(* Logix 5000 project; controller Todd_Test vendor 1 type 14 code 87 rev 20.19; software revision 20.04 *)

TASK MainTask (continuous, watchdog 500 ms) : MainProgram

MODULES
   Controller : vendor 1 type 14 code 87 (CompactLogixL23E_QB1_Controller 0, rev 20.19)
      LocalENB : vendor 1 type 12 code 190 (CompactLogixL23E_QB1_Ethernet 1, rev 20.11)
      Local : CompactBus (CompactVirtualAdapter 3, rev 20.11)
         Discrete_Inputs : vendor 1 type 7 code 320 (Compact 1, rev 3.1, Input RPI 20 ms)
         Discrete_Outputs : vendor 1 type 7 code 322 (Compact 2, rev 3.1, Output RPI 20 ms)
END_MODULES

TYPE ac_JobData :
STRUCT
   NoOperation : BOOL;
   Valid : BOOL;
   Invalid : BOOL;
   MisMatch : BOOL;
   Prompt : BOOL;
   OneShot : INT;
   Offset : DINT;
   HMIOffsetSelect : DINT;
   PartCode : DINT;
   License_Batch : STRING;
   Enable : z_HMIStylePBs;
   Data : z_Data;
END_STRUCT
END_TYPE

TYPE BEP_BS1 :
STRUCT
   License_Batch : STRING;
   PartCode : DINT;
   Handshake : DINT;
   FaultStatus : DINT;
END_STRUCT
END_TYPE

TYPE BS1_BEP :
STRUCT
   License_Batch : STRING;
   Type_ID : DINT;
   Handshake : DINT;
   FaultStatus : DINT;
END_STRUCT
END_TYPE

TYPE dt_Data_Track :
STRUCT
   DataGT0 : BOOL;
   PPCurrent : BOOL;
   NPPCurrent : BOOL;
   PEN : BOOL;
   NEQPrev : BOOL;
   MDTBuffer : BOOL;
   MDTNext : BOOL;
   Move : BOOL;
   MoveDat2PRev : BOOL;
   Move0toNext : BOOL;
   InputWord : DINT;
   OutputWord : DINT;
END_STRUCT
END_TYPE

TYPE dt_DataTrack :
STRUCT
   NoProc : BOOL;
   NoParts : BOOL;
   NoData : BOOL;
END_STRUCT
END_TYPE

TYPE dt_Prelims :
STRUCT
   BuffDat : BOOL;
   InitDat : BOOL;
   StaDat : BOOL;
   PrevDat : BOOL;
   NextDat : BOOL;
   MTBuff : BOOL;
END_STRUCT
END_TYPE

TYPE int_FromConveyor :
STRUCT
   Hearbeat : BOOL;
   PartPresent : BOOL;
   DataPresent : BOOL;
   CleartoExit : BOOL;
   BypassPart : BOOL;
   ComsGood : BOOL;
   SpareBool_2 : BOOL;
   SpareBool_3 : BOOL;
   SpareBool_4 : BOOL;
   PartCode : DINT;
   SpareDINT : DINT;
END_STRUCT
END_TYPE

TYPE int_ToConveyor :
STRUCT
   Heartbeat : BOOL;
   ReadytoReceiveAssembly : BOOL;
   ReadytoReceivePartCode : BOOL;
   PartCodeReceived : BOOL;
   PartReceivedACK : BOOL;
   ReadytoExit : BOOL;
   GoodPart : BOOL;
   RejectPart : BOOL;
   Partpresent_1 : BOOL;
   Partpresent_2 : BOOL;
   Partpresent_3 : BOOL;
   comsgood : BOOL;
   AutoMode : BOOL;
   ManualMode : BOOL;
   SpareBool_4 : BOOL;
   LastPart : DINT;
   CurrentPart : DINT;
END_STRUCT
END_TYPE

TYPE PF52x_I :
STRUCT
   DriveStatus : INT;
   Ready : BOOL;
   Active : BOOL;
   CommandDir : BOOL;
   ActualDir : BOOL;
   Accelerating : BOOL;
   Decelerating : BOOL;
   Faulted : BOOL;
   AtReference : BOOL;
   CommFreqCnt : BOOL;
   CommLogicCnt : BOOL;
   ParmsLocked : BOOL;
   DigIn1Active : BOOL;
   DigIn2Active : BOOL;
   DigIn3Active : BOOL;
   DigIn4Active : BOOL;
   OutputFreq : INT;
END_STRUCT
END_TYPE

TYPE PF52x_O :
STRUCT
   LogicCommand : INT;
   Stop : BOOL;
   Start : BOOL;
   Jog : BOOL;
   ClearFaults : BOOL;
   Forward : BOOL;
   Reverse : BOOL;
   ForceKeypadCtrl : BOOL;
   MOPIncrement : BOOL;
   AccelRate1 : BOOL;
   AccelRate2 : BOOL;
   DecelRate1 : BOOL;
   DecelRate2 : BOOL;
   FreqSel01 : BOOL;
   FreqSel02 : BOOL;
   FreqSel03 : BOOL;
   MOPDecrement : BOOL;
   FreqCommand : INT;
END_STRUCT
END_TYPE

TYPE u_AccuracyBalanceSequence :
STRUCT
   SpinCount : COUNTER;
   ReSpinDwell : TIMER;
   SequenceStep : u_TireBalanceAccuracySteps;
   OneShot : BOOL[32];
END_STRUCT
END_TYPE

TYPE u_ActionAdvanceReturn :
STRUCT
   Advance : up_ActionNew;
   Return : up_ActionNew;
END_STRUCT
END_TYPE

TYPE u_ActionCloseOpen :
STRUCT
   Close : up_ActionNew;
   Open : up_ActionNew;
END_STRUCT
END_TYPE

TYPE u_ActionEngDiseng :
STRUCT
   Engage : up_ActionNew;
   Disengage : up_ActionNew;
END_STRUCT
END_TYPE

TYPE u_ActionInflate :
STRUCT
   Comp : BOOL;
   ProcComp : BOOL;
   Auto : BOOL;
   AutoSetup : BOOL;
   Clear : BOOL;
   ClrSetup : BOOL;
   OutPwr : BOOL;
   Cmd : BOOL;
   Out : BOOL;
   Mem : BOOL;
   PB : BOOL;
   FLT : BOOL;
   Active : BOOL;
   EnableSkip : BOOL;
   EnableBypass : BOOL;
   Bypassed : BOOL;
   Prompt : BOOL;
   OutPwrPrompt : BOOL;
   AtBeadSeat : BOOL;
   BeadSeatProcessComp : BOOL;
   Setup3 : BOOL;
   Setup4 : BOOL;
   AntiRept : BOOL;
   OneShot : BOOL;
   Text : DINT;
   StatusType : DINT;
   SeatTMR : TIMER;
   FaultTMR : TIMER;
   TestTMR : TIMER;
END_STRUCT
END_TYPE

TYPE u_ActionInflateDeflate :
STRUCT
   Inflate : u_ActionInflate;
   Deflate : up_ActionNew;
END_STRUCT
END_TYPE

TYPE u_ActionInOut :
STRUCT
   In : up_ActionNew;
   Out : up_ActionNew;
END_STRUCT
END_TYPE

TYPE u_ActionLower4Raise :
STRUCT
   LowerToLock : up_ActionNew;
   LowerToChanger : up_ActionNew;
   LowerToJoin_1 : up_ActionNew;
   LowerToJoin_2 : up_ActionNew;
   Raise : up_ActionNew;
END_STRUCT
END_TYPE

TYPE u_ActionRaiseLower :
STRUCT
   Raise : up_ActionNew;
   Lower : up_ActionNew;
END_STRUCT
END_TYPE

TYPE u_ActionRetractExtend :
STRUCT
   Retract : up_ActionNew;
   Extend : up_ActionNew;
END_STRUCT
END_TYPE

TYPE u_BalanceGainCalSeq :
STRUCT
   SequenceStep : u_TireBalanceGainSteps;
   OneShot : BOOL[32];
END_STRUCT
END_TYPE

TYPE u_BalanceToolingCalibrationSequence :
STRUCT
   SequenceStep : u_TireBalanceToolCalSteps;
   OneShot : BOOL[32];
   CycleCounter : COUNTER;
   IndexAngle : REAL;
END_STRUCT
END_TYPE

TYPE u_StaMode :
STRUCT
   AutoReqAntiRpt : BOOL;
   AutoRdy : BOOL;
   Auto : BOOL;
   ExtrnAutoRdy : BOOL;
   Man : BOOL;
   Calibration : BOOL;
   ByPass : BOOL;
   BatchMode : BOOL;
   Tryout : BOOL;
END_STRUCT
END_TYPE

TYPE u_StaMode_BeadSeat :
STRUCT
   AutoReqAntiRpt : BOOL;
   AutoRdy : BOOL;
   Auto : BOOL;
   ExtrnAutoRdy : BOOL;
   Man : BOOL;
   TryOut : BOOL;
   ByPass : BOOL;
END_STRUCT
END_TYPE

TYPE u_TBAL_BALCycle :
STRUCT
   Action : up_ActionNew;
   Seq : u_TBAL_BALSteps;
   ChargeAmpDwell : TIMER;
   SampleDelay : TIMER;
   SpinDwell : TIMER;
   ChargeAmp : up_Relay;
   OneShot : BOOL[32];
END_STRUCT
END_TYPE

TYPE u_TBAL_BALSteps :
STRUCT
   EnableChargeAmplifier : BOOL;
   StartRotation : BOOL;
   SpindleAtSpeed : BOOL;
   StartSample : BOOL;
   SampleComplete : BOOL;
   StopAtAngle : BOOL;
   CorrectStopPosition : BOOL;
   CycleComplete : BOOL;
END_STRUCT
END_TYPE

TYPE u_TireBalanceAccuracySteps :
STRUCT
   CloseCentering : BOOL;
   LowerLifter : BOOL;
   OpenCentering : BOOL;
   LowerUpperTooling : BOOL;
   LockLowerTooling : BOOL;
   UnlockUpperTooling : BOOL;
   InflateTire : BOOL;
   PromptForEmptySpin : BOOL;
   StartBalanceEmpty : BOOL;
   PromptOpenDoorCouple : BOOL;
   PromptCoupleWeights : BOOL;
   PromptCoupleSpin : BOOL;
   StartCoupleSpin : BOOL;
   PromptOpenDoorStatic : BOOL;
   PrmptStaticWeights : BOOL;
   PromptForStaticSpin : BOOL;
   StartStaticSpin : BOOL;
   PromptOpenDoorLower : BOOL;
   PromptLowerWeight : BOOL;
   PromptForLowerSpin : BOOL;
   StartLowerSpin : BOOL;
   PromptOpenDoorUpper : BOOL;
   PromptUpperWeight : BOOL;
   PromptForUpperSpin : BOOL;
   StartUpperSpin : BOOL;
   PromptRemoveWeights : BOOL;
   PromptTestComplete : BOOL;
   DeflateTire : BOOL;
   LockUpperTooling : BOOL;
   ExtendBeadBreaker : BOOL;
   UnlockLowerTooling : BOOL;
   RaiseUpperTooling : BOOL;
   RaiseLifter : BOOL;
   RaiseBeadBreaker : BOOL;
   AccuracyTestComplete : BOOL;
END_STRUCT
END_TYPE

TYPE u_TireBalanceGainSteps :
STRUCT
   CloseCentering : BOOL;
   LowerLifter : BOOL;
   OpenCentering : BOOL;
   LowerUpperTooling : BOOL;
   LockLowerTooling : BOOL;
   UnlockUpperTooling : BOOL;
   InflateTire : BOOL;
   PromptForEmptySpin : BOOL;
   StartBalanceEmpty : BOOL;
   PromptOpenDoorUpper : BOOL;
   PromptUpperWeight : BOOL;
   PromptForUpperSpin : BOOL;
   StartBalanceUpper : BOOL;
   PromptOpenDoorLower : BOOL;
   PromptLowerWeight : BOOL;
   PromptForLowerSpin : BOOL;
   StartBalanceLower : BOOL;
   PromptOpenDoorEmpty : BOOL;
   PromptRemoveWeights : BOOL;
   DeflateTire : BOOL;
   LockUpperTooling : BOOL;
   ExtendBeadBreakers : BOOL;
   UnlockLowerTooling : BOOL;
   RaiseUpperTooling : BOOL;
   RaiseLifter : BOOL;
   RaiseBeadBreakers : BOOL;
   GainCalibrationComplete : BOOL;
END_STRUCT
END_TYPE

TYPE u_TireBalanceToolCalSteps :
STRUCT
   CloseCentering : BOOL;
   LowerLifter : BOOL;
   OpenCentering : BOOL;
   LowerUpperTooling : BOOL;
   LockLowerTooling : BOOL;
   UnlockUpperTooling : BOOL;
   InflateTire : BOOL;
   StartBalance : BOOL;
   DeflateTire : BOOL;
   LockUpperTooling : BOOL;
   AdvanceBeadBreakers : BOOL;
   UnlockLowerTooling : BOOL;
   RaiseUpperTooling : BOOL;
   IndexTireToNextAngle : BOOL;
   RaiseLifter : BOOL;
   RaiseBeadBreaker : BOOL;
   AlignTooling : BOOL;
END_STRUCT
END_TYPE

TYPE uc_BDS_XFRIntlk :
STRUCT
   Auto : BOOL;
   Man : BOOL;
   AtLoad : BOOL;
   AtUnload : BOOL;
   Bypass : BOOL;
   ByPassAllowed : BOOL;
   InPosition : BOOL;
   NextConvFull : BOOL;
   LeavingPX : BOOL;
   Load_Unload : BOOL;
   DriveOK : BOOL;
   HiSpdEn : BOOL;
   DrvRunningFwd : BOOL;
   DrvRunningRev : BOOL;
   TWRunAudit : BOOL;
   PrimaryBalanceMode : BOOL;
   RdytoExitFwd : BOOL;
   RdytoExitRev : BOOL;
   RdytoExitSide : BOOL;
   RequestNextPart : BOOL;
   ClrtoEnterFwd : BOOL;
   ClrtoEnterRev : BOOL;
   ClrtoEnterSide : BOOL;
   JobinTransitFwd : BOOL;
   JobinTransitRev : BOOL;
   JobinTransitSide : BOOL;
   IndexInPB : BOOL;
   IndexOutPB : BOOL;
   RevInPB : BOOL;
   RevOutPB : BOOL;
   BalanceSampleComplete : BOOL;
   ValidModel : BOOL;
   MachineEmpty : BOOL;
   NoSkidPres : BOOL;
   Heartbeat : BOOL;
END_STRUCT
END_TYPE

TYPE uc_BeadSeaterServoTargets :
STRUCT
   PressUnitAdvanced : REAL;
   PressUnitReturned : REAL;
   UpperUnitAdvanced : REAL;
   LowerUnitAdvanced : REAL;
   UpperRollerAdvanced : REAL;
   LowerRollerAdvanced : REAL;
   LifterMidPosition : REAL;
   LifterLowerPosition : REAL;
END_STRUCT
END_TYPE

TYPE uc_BeadSeaterServoTargetsWithTorque :
STRUCT
   PressUnitAdvanced : REAL;
   PressUnitReturned : REAL;
   UpperUnitAdvanced : REAL;
   LowerUnitAdvanced : REAL;
   UpperRollerAdvanced : REAL;
   UpperRollerAdvanceLowTorqueLimit : REAL;
   UpperRollerAdvanceHighTorqueLimit : REAL;
   UpperRollerAdvanceMinTorqueApplied : REAL;
   UpperRollerAdvanceMaxTorqueApplied : REAL;
   LowerRollerAdvanced : REAL;
   LowerRollerAdvanceLowTorqueLimit : REAL;
   LowerRollerAdvanceHighTorqueLimit : REAL;
   LowerRollerAdvanceMinTorqueApplied : REAL;
   LowerRollerAdvanceMaxTorqueApplied : REAL;
   LifterMidPosition : REAL;
   LifterLowerPosition : REAL;
END_STRUCT
END_TYPE

TYPE uc_Gripper :
STRUCT
   GripTorque : REAL;
   GripSpeed : REAL;
   RelaxSpeed : REAL;
   RelaxOffset : REAL;
END_STRUCT
END_TYPE

TYPE uc_Home :
STRUCT
   HomingTorque : REAL;
   Offset : REAL;
   Velocity : REAL;
END_STRUCT
END_TYPE

TYPE uc_Job :
STRUCT
   TWStatus : uc_TWStatus;
   TWModel : uc_TWModel;
   TWCorrection : uc_TWCorrection;
   Xfer : uc_BDS_XFRIntlk;
END_STRUCT
END_TYPE

TYPE uc_Job_BC :
STRUCT
   TWStatus : uc_TWStatus;
   TWModel : uc_TWModel;
   TWCorrection : uc_TWCorrection;
   Xfer : uc_BDS_XFRIntlk;
   BarCode : SINT[80];
END_STRUCT
END_TYPE

TYPE uc_KokusaiModelData :
STRUCT
   Name : STRING;
   WheelDiam : DINT;
   WheelWidth : DINT;
   WheelOffset : DINT;
   OutsideDiameter : DINT;
   PressStroke : DINT;
   Bypass : BOOL;
   Servo : uc_BeadSeaterServoTargets;
   RotateTime : DINT;
END_STRUCT
END_TYPE

TYPE uc_KokusaiModelDataWithTorque :
STRUCT
   Type_ID : DINT;
   WheelDiam : DINT;
   WheelWidth : DINT;
   WheelOffset : DINT;
   OutsideDiameter : REAL;
   PressStroke : DINT;
   Bypass : BOOL;
   Servo : uc_BeadSeaterServoTargetsWithTorque;
   RotateTime : DINT;
END_STRUCT
END_TYPE

TYPE uc_KokusaiModelTorqueData :
STRUCT
   LowerRollerAdvanceTorqueApplied : REAL[101];
   LowerRollerRotatingMinTorqueApplied : REAL[101];
   LowerRollerRotatingMaxTorqueApplied : REAL[101];
   LowerRollerRotatingAveTorqueApplied : REAL[101];
   UpperRollerAdvanceTorqueApplied : REAL[101];
   UpperRollerRotatingMinTorqueApplied : REAL[101];
   UpperRollerRotatingMaxTorqueApplied : REAL[101];
   UpperRollerRotatingAveTorqueApplied : REAL[101];
END_STRUCT
END_TYPE

TYPE uc_TransferInterlock :
STRUCT
   Auto : BOOL;
   Man : BOOL;
   AtLoad : BOOL;
   AtUnload : BOOL;
   Bypass : BOOL;
   InPosition : BOOL;
   NextConvFull : BOOL;
   LeavingPX : BOOL;
   Spare8 : BOOL;
   DriveOK : BOOL;
   HiSpdEn : BOOL;
   DrvRunningFwd : BOOL;
   DrvRunningRev : BOOL;
   Spare13 : BOOL;
   Spare14 : BOOL;
   RdytoExitFwd : BOOL;
   RdytoExitRev : BOOL;
   RdytoExitSide : BOOL;
   ClrtoEnterFwd : BOOL;
   ClrtoEnterRev : BOOL;
   ClrtoEnterSide : BOOL;
   JobinTransitFwd : BOOL;
   JobinTransitRev : BOOL;
   JobinTransitSide : BOOL;
   IndexInPB : BOOL;
   IndexOutPB : BOOL;
   RevInPB : BOOL;
   RevOutPB : BOOL;
   Spare28 : BOOL;
   Spare29 : BOOL;
   MachineEmpty : BOOL;
   NoSkidPres : BOOL;
   Heartbeat : DINT;
   BEP_BS1_ComboRdyToReceive : BOOL;
   BEP_BS1_ComboReceived : BOOL;
   BEP_BS1_ComboDataMismatch : BOOL;
   BEP_BS1_BypassStation : BOOL;
   BEP_BS1_RejectAssy : BOOL;
   BS1_BEP_ComboSent : BOOL;
   BS1_BEP_ComboReceived : BOOL;
   BS1_BEP_NotTested : BOOL;
   BS1_BEP_PartPresent : BOOL;
   BS1_BEP_ComboDataMismatch : BOOL;
   BS1_BEP_CheckTireMode : BOOL;
   ComboRdyToReceive : BOOL;
END_STRUCT
END_TYPE

TYPE uc_TransferInterlock_New :
STRUCT
   Auto : BOOL;
   Man : BOOL;
   AtLoad : BOOL;
   AtUnload : BOOL;
   Bypass : BOOL;
   InPosition : BOOL;
   NextConvFull : BOOL;
   LeavingPX : BOOL;
   AdapterOKForNext : BOOL;
   DriveOK : BOOL;
   HiSpdEn : BOOL;
   DrvRunningFwd : BOOL;
   DrvRunningRev : BOOL;
   AdapterOKForCurrent : BOOL;
   RequestNextPart : BOOL;
   RdytoExitFwd : BOOL;
   RdytoExitRev : BOOL;
   RdytoExitSide : BOOL;
   TransferedDataFwd : BOOL;
   TransferedDataRev : BOOL;
   TransferedDataSide : BOOL;
   ClrToEnterFwd : BOOL;
   ClrToEnterRev : BOOL;
   ClrToEnterSide : BOOL;
   JobinTransitFwd : BOOL;
   JobinTransitRev : BOOL;
   JobinTransitSide : BOOL;
   IndexInPB : BOOL;
   IndexOutPB : BOOL;
   RevInPB : BOOL;
   RevOutPB : BOOL;
   Spare28 : BOOL;
   Spare29 : BOOL;
   Spare30 : BOOL;
   NoSkidPres : BOOL;
   Heartbeat : DINT;
END_STRUCT
END_TYPE

TYPE uc_TWCorrection :
STRUCT
   BalanceStaticAmount : REAL;
   BalanceStaticAngle : DINT;
   BalanceCoupleAmount : REAL;
   BalanceCoupleAngle : DINT;
   PlaneUpperAmount : REAL;
   PlaneUpperAngle : DINT;
   PlaneLowerAmount : REAL;
   PlaneLowerAngle : DINT;
   UpperWeightAmount : REAL;
   UpperWeightAngle : DINT;
   UpperWeightStyle : DINT;
   LowerWeightAmount : REAL;
   LowerWeightAngle : DINT;
   LowerWeightStyle : DINT;
   ShortReachCorrection : DINT;
   SecondCorrection : DINT;
   FirstCorrection : DINT;
   UpperWeightRadius : DINT;
   LowerWeightRadius : DINT;
   UpperWeightHeight : DINT;
   LowerWeightHeight : DINT;
END_STRUCT
END_TYPE

TYPE uc_TWModel :
STRUCT
   PartCode : DINT;
   WheelDiameter : DINT;
   Desc0_1 : DINT;
   Desc2_3 : DINT;
   Desc4_5 : DINT;
   Desc6_7 : DINT;
   Desc8_9 : DINT;
   Desc10_11 : DINT;
   Desc12_13 : DINT;
   Desc14_15 : DINT;
   Desc16_17 : DINT;
   Desc18_19 : DINT;
   Key : DINT;
   TID : DINT;
END_STRUCT
END_TYPE

TYPE uc_TWStatus :
STRUCT
   GoodAssembly : BOOL;
   CorrectableAssembly : BOOL;
   UncorrectableAssembly : BOOL;
   ByPassAssembly : BOOL;
   MiniSpare : BOOL;
   Material : BOOL;
   MidPlaneApply : BOOL;
   UpSideDown : BOOL;
END_STRUCT
END_TYPE

TYPE uc_UFB_BALData :
STRUCT
   Rank : INT;
   MarkPattern : INT;
   SortPosition : INT;
   MarkAngle : INT;
   StaticAmount : REAL;
   StaticAmountUnits : INT;
   StaticAngle : INT;
   CoupleAmount : REAL;
   CoupleAmountUnits : INT;
   CoupleAngle : INT;
   UpperAmount : REAL;
   UpperAmountUnits : INT;
   UpperAngle : INT;
   LowerAmount : REAL;
   LowerAmountUnits : INT;
   LowerAngle : INT;
END_STRUCT
END_TYPE

TYPE uc_UFB_BALStatus :
STRUCT
   ByPass : BOOL;
   BALGainCalRequired : BOOL;
   BALToolCalRequired : BOOL;
   MeasureBAL : BOOL;
END_STRUCT
END_TYPE

TYPE uc_UFB_Data :
STRUCT
   Model : INT;
   RimStep : INT;
   Adapter : INT;
   BeadDiameter : INT;
   BeadWidth : INT;
   OutsideDiameter : INT;
   Weight : INT;
   RankFinal : INT;
   MarkPatternFinal : INT;
   SortPositionFinal : INT;
   SerialNumber : SINT[20];
   BAL : uc_UFB_BALData;
   RO : uc_UFB_ROData;
   LSU : uc_UFB_LSUData;
   HSU : uc_UFB_HSUData;
END_STRUCT
END_TYPE

TYPE uc_UFB_HSUData :
STRUCT
   Rank : INT;
   MarkPattern : INT;
   SortPosition : INT;
   MarkAngle : INT;
   LoadForce : INT;
   ConicityForce : INT;
   PlySteerForce : INT;
   SpeedRPM : INT;
   SurfaceVelocity : INT;
   RadialOverallAmountCW : INT;
   RadialOverallAngleCW : INT;
   Radial1stHarmonicAmountCW : INT;
   Radial1stHarmonicAngleCW : INT;
   Radial2ndHarmonicAmountCW : INT;
   Radial2ndHarmonicAngleCW : INT;
   Radial3rdHarmonicAmountCW : INT;
   Radial3rdHarmonicAngleCW : INT;
   Radial4thHarmonicAmountCW : INT;
   Radial4thHarmonicAngleCW : INT;
   Radial5thHarmonicAmountCW : INT;
   Radial5thHarmonicAngleCW : INT;
   RadialOverallAmountCCW : INT;
   RadialOverallAngleCCW : INT;
   Radial1stHarmonicAmountCCW : INT;
   Radial1stHarmonicAngleCCW : INT;
   Radial2ndHarmonicAmountCCW : INT;
   Radial2ndHarmonicAngleCCW : INT;
   Radial3rdHarmonicAmountCCW : INT;
   Radial3rdHarmonicAngleCCW : INT;
   Radial4thHarmonicAmountCCW : INT;
   Radial4thHarmonicAngleCCW : INT;
   Radial5thHarmonicAmountCCW : INT;
   Radial5thHarmonicAngleCCW : INT;
   LateralOverallAmountCW : INT;
   LateralOverallAngleCW : INT;
   Lateral1stHarmonicAmountCW : INT;
   Lateral1stHarmonicAngleCW : INT;
   Lateral2ndHarmonicAmountCW : INT;
   Lateral2ndHarmonicAngleCW : INT;
   Lateral3rdHarmonicAmountCW : INT;
   Lateral3rdHarmonicAngleCW : INT;
   Lateral4thHarmonicAmountCW : INT;
   Lateral4thHarmonicAngleCW : INT;
   Lateral5thHarmonicAmountCW : INT;
   Lateral5thHarmonicAngleCW : INT;
   LateralForceDeviationAmountCW : INT;
   LateralOverallAmountCCW : INT;
   LateralOverallAngleCCW : INT;
   Lateral1stHarmonicAmountCCW : INT;
   Lateral1stHarmonicAngleCCW : INT;
   Lateral2ndHarmonicAmountCCW : INT;
   Lateral2ndHarmonicAngleCCW : INT;
   Lateral3rdHarmonicAmountCCW : INT;
   Lateral3rdHarmonicAngleCCW : INT;
   Lateral4thHarmonicAmountCCW : INT;
   Lateral4thHarmonicAngleCCW : INT;
   Lateral5thHarmonicAmountCCW : INT;
   Lateral5thHarmonicAngleCCW : INT;
   LateralForceDeviationAmountCCW : INT;
   TangentialOverallAmountCW : INT;
   TangentialOverallAngleCW : INT;
   Tangential1stHarmonicAmountCW : INT;
   Tangential1stHarmonicAngleCW : INT;
   Tangential2ndHarmonicAmountCW : INT;
   Tangential2ndHarmonicAngleCW : INT;
   Tangential3rdHarmonicAmountCW : INT;
   Tangential3rdHarmonicAngleCW : INT;
   Tangential4thHarmonicAmountCW : INT;
   Tangential4thHarmonicAngleCW : INT;
   Tangential5thHarmonicAmountCW : INT;
   Tangential5thHarmonicAngleCW : INT;
   TangentialOverallAmountCCW : INT;
   TangentialOverallAngleCCW : INT;
   Tangential1stHarmonicAmountCCW : INT;
   Tangential1stHarmonicAngleCCW : INT;
   Tangential2ndHarmonicAmountCCW : INT;
   Tangential2ndHarmonicAngleCCW : INT;
   Tangential3rdHarmonicAmountCCW : INT;
   Tangential3rdHarmonicAngleCCW : INT;
   Tangential4thHarmonicAmountCCW : INT;
   Tangential4thHarmonicAngleCCW : INT;
   Tangential5thHarmonicAmountCCW : INT;
   Tangential5thHarmonicAngleCCW : INT;
END_STRUCT
END_TYPE

TYPE uc_UFB_Job :
STRUCT
   Data : uc_UFB_Data;
   Status : uc_UFB_Status;
END_STRUCT
END_TYPE

TYPE uc_UFB_LSUData :
STRUCT
   Rank : INT;
   MarkPattern : INT;
   SortPosition : INT;
   MarkAngle : INT;
   LoadForce : INT;
   ConicityForce : INT;
   PlySteerForce : INT;
   SpeedRPM : INT;
   SurfaceVelocity : INT;
   RadialOverallAmountCW : INT;
   RadialOverallAngleCW : INT;
   Radial1stHarmonicAmountCW : INT;
   Radial1stHarmonicAngleCW : INT;
   Radial2ndHarmonicAmountCW : INT;
   Radial2ndHarmonicAngleCW : INT;
   Radial3rdHarmonicAmountCW : INT;
   Radial3rdHarmonicAngleCW : INT;
   Radial4thHarmonicAmountCW : INT;
   Radial4thHarmonicAngleCW : INT;
   Radial5thHarmonicAmountCW : INT;
   Radial5thHarmonicAngleCW : INT;
   RadialOverallAmountCCW : INT;
   RadialOverallAngleCCW : INT;
   Radial1stHarmonicAmountCCW : INT;
   Radial1stHarmonicAngleCCW : INT;
   Radial2ndHarmonicAmountCCW : INT;
   Radial2ndHarmonicAngleCCW : INT;
   Radial3rdHarmonicAmountCCW : INT;
   Radial3rdHarmonicAngleCCW : INT;
   Radial4thHarmonicAmountCCW : INT;
   Radial4thHarmonicAngleCCW : INT;
   Radial5thHarmonicAmountCCW : INT;
   Radial5thHarmonicAngleCCW : INT;
   LateralOverallAmountCW : INT;
   LateralOverallAngleCW : INT;
   Lateral1stHarmonicAmountCW : INT;
   Lateral1stHarmonicAngleCW : INT;
   Lateral2ndHarmonicAmountCW : INT;
   Lateral2ndHarmonicAngleCW : INT;
   Lateral3rdHarmonicAmountCW : INT;
   Lateral3rdHarmonicAngleCW : INT;
   Lateral4thHarmonicAmountCW : INT;
   Lateral4thHarmonicAngleCW : INT;
   Lateral5thHarmonicAmountCW : INT;
   Lateral5thHarmonicAngleCW : INT;
   LateralForceDeviationAmountCW : INT;
   LateralOverallAmountCCW : INT;
   LateralOverallAngleCCW : INT;
   Lateral1stHarmonicAmountCCW : INT;
   Lateral1stHarmonicAngleCCW : INT;
   Lateral2ndHarmonicAmountCCW : INT;
   Lateral2ndHarmonicAngleCCW : INT;
   Lateral3rdHarmonicAmountCCW : INT;
   Lateral3rdHarmonicAngleCCW : INT;
   Lateral4thHarmonicAmountCCW : INT;
   Lateral4thHarmonicAngleCCW : INT;
   Lateral5thHarmonicAmountCCW : INT;
   Lateral5thHarmonicAngleCCW : INT;
   LateralForceDeviationAmountCCW : INT;
END_STRUCT
END_TYPE

TYPE uc_UFB_MEAStatus :
STRUCT
   ByPass : BOOL;
   ROToolCalRequired : BOOL;
   LSUToolCalRequired : BOOL;
   MeasureRO : BOOL;
   ROMeasureType : INT;
   MeasureLSU : BOOL;
   LSU_SingleDirection : BOOL;
   LSU_CWDirection : BOOL;
   EnglishUnits : BOOL;
END_STRUCT
END_TYPE

TYPE uc_UFB_ROData :
STRUCT
   Rank : INT;
   MarkPattern : INT;
   SortPosition : INT;
   MarkAngle : INT;
   RadialTopPeakAmount : INT;
   RadialTopPeakAngle : INT;
   RadialTop1stAmount : INT;
   RadialTop1stAngle : INT;
   RadialTop2ndAmount : INT;
   RadialTop2ndAngle : INT;
   RadialCenterPeakAmount : INT;
   RadialCenterPeakAngle : INT;
   RadialCenter1stAmount : INT;
   RadialCenter1stAngle : INT;
   RadialCenter2ndAmount : INT;
   RadialCenter2ndAngle : INT;
   RadialBottomPeakAmount : INT;
   RadialBottomPeakAngle : INT;
   RadialBottom1stAmount : INT;
   RadialBottom1stAngle : INT;
   RadialBottom2ndAmount : INT;
   RadialBottom2ndAngle : INT;
   LateralTopPeakAmount : INT;
   LateralTopPeakAngle : INT;
   LateralTop1stAmount : INT;
   LateralTop1stAngle : INT;
   LateralTop2ndAmount : INT;
   LateralTop2ndAngle : INT;
   LateralBottomPeakAmount : INT;
   LateralBottomPeakAngle : INT;
   LateralBottom1stAmount : INT;
   LateralBottom1stAngle : INT;
   LateralBottom2ndAmount : INT;
   LateralBottom2ndAngle : INT;
   TopBulgeAmount : INT;
   TopBulgeAngle : INT;
   TopDentAmount : INT;
   TopDentAngle : INT;
   BottomBulgeAmount : INT;
   BottomBulgeAngle : INT;
   BottomDentAmount : INT;
   BottomDentAngle : INT;
END_STRUCT
END_TYPE

TYPE uc_UFB_Status :
STRUCT
   ByPass : BOOL;
   CertificationMode : BOOL;
   UpSideDown : BOOL;
   MEA : uc_UFB_MEAStatus;
   BAL : uc_UFB_BALStatus;
END_STRUCT
END_TYPE

TYPE ud_KokusaiServoConstants :
STRUCT
   cForward : DINT;
   cReverse : DINT;
   cPercentMaxSpeed : DINT;
   cDisabled : DINT;
   cEnabled : DINT;
   cAbsolute : DINT;
   cIncremental : DINT;
   cRotaryShortestPath : DINT;
   cRotaryPositive : DINT;
   cRotaryNegative : DINT;
   cAbsoluteMasterOffset : DINT;
   cIncrementalMasterOffset : DINT;
   cTourqueLimit : ud_KokusaiServoTorqueContants;
END_STRUCT
END_TYPE

TYPE ud_KokusaiServoTorqueContants :
STRUCT
   Axis1 : REAL;
   Axis2 : REAL;
   Axis3 : REAL;
   Axis4 : REAL;
   Axis5 : REAL;
   Axis6 : REAL;
   Axis7 : REAL;
   Axis8 : REAL;
   Axis9 : REAL;
   Axis10 : REAL;
   Axis11 : REAL;
   Axis12 : REAL;
   Axis13 : REAL;
   Axis14 : REAL;
   Axis15 : REAL;
END_STRUCT
END_TYPE

TYPE ud_KokusaiTransferGripper :
STRUCT
   InPositionLowRangeLimit : DINT;
   InPositionHighRangeLimit : DINT;
   Model : ud_KokusaiTransferGripperModel[10000];
END_STRUCT
END_TYPE

TYPE ud_KokusaiTransferGripperModel :
STRUCT
   GripperClosedPositionHighSafety : DINT;
   GripperClosedPosition : REAL;
   GripperOpenedPositionHighSafety : DINT;
   GripperOpenedPosition : REAL;
END_STRUCT
END_TYPE

TYPE udt_AutomaticAutoStop :
STRUCT
   PP_CenteringConveyor : BOOL;
   PP_BeadSeaterStation : BOOL;
   Engaged : BOOL;
   Complete : BOOL;
   SpareBool_01 : BOOL;
   SpareBool_02 : BOOL;
   SpareBool_03 : BOOL;
   SpareBool_04 : BOOL;
   ONS : INT;
   SpareDint : DINT;
   EngageTimer : TIMER;
END_STRUCT
END_TYPE

TYPE udt_PanelViewButton :
STRUCT
   Enable_PVPB : BOOL;
   Enabled_PVLT : BOOL;
   EnabledInternal : BOOL;
   ONS : BOOL;
END_STRUCT
END_TYPE

TYPE up_ActionNew :
STRUCT
   Comp : BOOL;
   ProcComp : BOOL;
   Auto : BOOL;
   AutoSetup : BOOL;
   ClrSetup : BOOL;
   ClearStart : BOOL;
   ClearThru : BOOL;
   OutPwr : BOOL;
   Cmd : BOOL;
   Out : BOOL;
   Mem : BOOL;
   PB : BOOL;
   FLT : BOOL;
   Active : BOOL;
   EnableSkip : BOOL;
   EnableBypass : BOOL;
   Bypassed : BOOL;
   Prompt : BOOL;
   OutPwrPrompt : BOOL;
   Setup1 : BOOL;
   Setup2 : BOOL;
   Setup3 : BOOL;
   Setup4 : BOOL;
   AntiRept : BOOL;
   OneShot : BOOL[32];
   TMR : TIMER[5];
   FaultTMR : TIMER;
END_STRUCT
END_TYPE

TYPE up_BalanceLifter :
STRUCT
   Command : up_BalanceLifterCommands;
   Status : up_BalanceLifterStatus;
   MidPositionDwell : TIMER;
   EnableMotion : BOOL;
   RaiseTargetIsValid : BOOL;
   MiddleTargetIsValid : BOOL;
   LowerTargetIsValid : BOOL;
   RaisedPositionTarget : REAL;
   RaisedLowLimit : REAL;
   RaisedHighLimit : REAL;
   MiddlePositionTarget : REAL;
   MiddleLowLimit : REAL;
   MiddleHighLimit : REAL;
   MiddleLowSafety : REAL;
   MiddleHighSafety : REAL;
   LowerPositionTarget : REAL;
   LowerLowLimit : REAL;
   LowerHighLimit : REAL;
   LowerLowSafety : REAL;
   LowerHighSafety : REAL;
   JogSpeedPercent : DINT;
END_STRUCT
END_TYPE

TYPE up_BalanceLifterCommands :
STRUCT
   JogMode : BOOL;
   JogLifterDown : BOOL;
   JogLifterUp : BOOL;
   StartHomePulse : BOOL;
   HomeLifterServo : BOOL;
   SetLifterRaisedPosition : BOOL;
   SetLifterLoweredCalibration : BOOL;
   SetLifterMiddlePosition : BOOL;
   SetLifterLoweredPosition : BOOL;
END_STRUCT
END_TYPE

TYPE up_BalanceLifterStatus :
STRUCT
   AtHomePosition : BOOL;
   ValidRaisedPosition : BOOL;
   ValidMiddlePosition : BOOL;
   ValidLoweredPosition : BOOL;
END_STRUCT
END_TYPE

TYPE up_BalanceSpindleServo :
STRUCT
   Command : up_SpindleServoCommands;
   Status : up_SpindleServoStatus;
   EnableMotion : BOOL;
   StartHomeSearch : BOOL;
   SearchForSpindleHome : BOOL;
   RetrySetHome : BOOL;
   VelocityInRange : BOOL;
   AtBalanceSpeed : BOOL;
   AtRunoutSpeed : BOOL;
   RimChangeAngleValid : BOOL;
   RimUnlockAngleValid : BOOL;
   MarkerAngle : REAL;
   OrientTargetAngle : REAL;
   OrientTargetHighLimit : REAL;
   OrientTargetLowLimit : REAL;
   MaxVelocityError : REAL;
   UpperFaultSpeed : REAL;
   LowerFaultSpeed : REAL;
   UpperToolingAngle : REAL;
   UpperToolingHighLimit : REAL;
   UpperToolingLowLimit : REAL;
   UpperToolingAlignmentTarget : REAL;
   UpperToolingAlignmentError : REAL;
   JogSpeed : REAL;
   OrientSpeed : REAL;
   RunoutSpeed : REAL;
   RunoutSpeedHigh : REAL;
   RunoutSpeedLow : REAL;
   BalanceSpeed : REAL;
   BalanceSpeedHigh : REAL;
   BalanceSpeedLow : REAL;
   AccelRate : REAL;
   DecelRate : REAL;
   BalanceRevolutions : DINT;
   BalanceDistance : REAL;
   RunoutRevolutions : DINT;
   RunoutDistance : REAL;
   SpindleStartAngle : REAL;
   SpindleSlipAngle : REAL;
   FailsafeTimer : TIMER;
   RimChangerAngleTarget : REAL;
   RimChangerHighLimit : REAL;
   RimChangerLowLimit : REAL;
   RimChangeValidHighLimit : REAL;
   RimChangeValidLowLimit : REAL;
   RimUnlockAngleTarget : REAL;
   RimUnlockHighLimit : REAL;
   RimUnlockLowLimit : REAL;
   RimUnlockValidHighLimit : REAL;
   RimUnlockValidLowLimit : REAL;
END_STRUCT
END_TYPE

TYPE up_ConveyorServo :
STRUCT
   EnableMotion : BOOL;
   MoveInLength : REAL;
   MoveOutLength : REAL;
END_STRUCT
END_TYPE

TYPE up_ConveyorWidthServo :
STRUCT
   Command : up_ConveyorWidthServoCommands;
   Status : up_ConveyorWidthServoStatus;
   EnableMotion : BOOL;
   AdapterTargetValid : BOOL;
   TransferTargetValid : BOOL;
   AdapterPositionTarget : REAL;
   AdapterPositionHiLimit : REAL;
   AdapterPositionLoLimit : REAL;
   TransferPositionTarget : REAL;
   TransferPositionHiLimit : REAL;
   TransferPositionLoLimit : REAL;
   JogSpeedPercent : DINT;
END_STRUCT
END_TYPE

TYPE up_ConveyorWidthServoCommands :
STRUCT
   JogMode : BOOL;
   JogClose : BOOL;
   JogOpen : BOOL;
   StartHomePulse : BOOL;
   HomeServo : BOOL;
END_STRUCT
END_TYPE

TYPE up_ConveyorWidthServoStatus :
STRUCT
   HomePosition : BOOL;
   ValidAdapterPosition : BOOL;
   ValidTransferPosition : BOOL;
END_STRUCT
END_TYPE

TYPE up_Cycle :
STRUCT
   InCycle : BOOL;
   AllPartsLoaded : BOOL;
   Finished : BOOL;
   FirstAutoCycle : BOOL;
   LoadPosition : BOOL;
   NoPartsLoaded : BOOL;
   NoProcComp : BOOL;
   NoProcInit : BOOL;
   NoStepsComp : BOOL;
   ProcComp : BOOL;
   ResetProcComp : BOOL;
   Resume : BOOL;
   RetToLoad : BOOL;
   RetToUnload : BOOL;
   SetProcComp : BOOL;
   Start : BOOL;
   Started : BOOL;
   StepsComp : BOOL;
   UnLoadPosition : BOOL;
   WaitingForLoad : BOOL;
   Idle : TIMER;
END_STRUCT
END_TYPE

TYPE up_Cylinder :
STRUCT
   PX1 : BOOL;
   PX1NOnFlt : BOOL;
   PX1NOffFlt : BOOL;
   BypPX1NOn : BOOL;
   BypPX1NOff : BOOL;
   PX2 : BOOL;
   PX2NOnFlt : BOOL;
   PX2NOffFlt : BOOL;
   BypPX2NOn : BOOL;
   BypPX2NOff : BOOL;
END_STRUCT
END_TYPE

TYPE up_CylinderBackToBack :
STRUCT
   PX1 : BOOL;
   PX1NOnFlt : BOOL;
   PX1NOffFlt : BOOL;
   BypPX1NOn : BOOL;
   BypPX1NOff : BOOL;
   PX2 : BOOL;
   PX2NOnFlt : BOOL;
   PX2NOffFlt : BOOL;
   BypPX2NOn : BOOL;
   BypPX2NOff : BOOL;
   PX3 : BOOL;
   PX3NOnFlt : BOOL;
   PX3NOffFlt : BOOL;
   BypPX3NOn : BOOL;
   BypPX3NOff : BOOL;
   PX4 : BOOL;
   PX4NOnFlt : BOOL;
   PX4NOffFlt : BOOL;
   BypPX4NOn : BOOL;
   BypPX4NOff : BOOL;
END_STRUCT
END_TYPE

TYPE up_Motion5Position :
STRUCT
   PX1 : BOOL;
   PX2 : BOOL;
   PX3 : BOOL;
   PX4 : BOOL;
   PX5 : BOOL;
END_STRUCT
END_TYPE

TYPE up_Part :
STRUCT
   Pres : BOOL;
   NotPres : BOOL;
   PresSwitches : BOOL;
   NotPresSwitches : BOOL;
   PresMemory : BOOL;
   Sw1NotOff : BOOL;
   Sw2NotOff : BOOL;
   Sw3NotOff : BOOL;
   Sw4NotOff : BOOL;
   Sw5NotOff : BOOL;
   Sw6NotOff : BOOL;
   Sw1NotOn : BOOL;
   Sw2NotOn : BOOL;
   Sw3NotOn : BOOL;
   Sw4NotOn : BOOL;
   Sw5NotOn : BOOL;
   Sw6NotOn : BOOL;
   LoadedProp : BOOL;
   LoadPosn : BOOL;
   Load : up_ActionNew;
   TryoutPresent : TIMER;
   TryoutNotPresent : TIMER;
END_STRUCT
END_TYPE

TYPE up_Relay :
STRUCT
   DiagEnable : BOOL;
   FltedOnMem : BOOL;
   Input : BOOL;
   Mimic : BOOL;
   Output : BOOL;
   FltTim : TIMER;
   OnTim : TIMER;
END_STRUCT
END_TYPE

TYPE up_RunoutServo :
STRUCT
   Command : up_RunoutServoCommands;
   Status : up_RunoutServoStatus;
   EnableMotion : BOOL;
   TargetIsValid : BOOL;
   Target : REAL;
   JogSpeedPercent : DINT;
   TargetHighLimit : REAL;
   TargetLowLimit : REAL;
END_STRUCT
END_TYPE

TYPE up_RunoutServoCommands :
STRUCT
   JogMode : BOOL;
   JogFoward : BOOL;
   JogReverse : BOOL;
   StartHomePulse : BOOL;
   HomeServo : BOOL;
END_STRUCT
END_TYPE

TYPE up_RunoutServoStatus :
STRUCT
   AtHomePosition : BOOL;
END_STRUCT
END_TYPE

TYPE up_ServoAdvanceReturn :
STRUCT
   Command : up_ServoAdvanceReturnCommands;
   Status : up_ServoAdvanceReturnStatus;
   EnableMotion : BOOL;
   ReturnedTargetIsValid : BOOL;
   AdvancedTargetIsValid : BOOL;
   ReturnedPositionTarget : REAL;
   ReturnedLowLimit : REAL;
   ReturnedHighLimit : REAL;
   ReturnedLowSafety : REAL;
   ReturnedHighSafety : REAL;
   AdvancedPositionTarget : REAL;
   AdvancedLowLimit : REAL;
   AdvancedHighLimit : REAL;
   AdvancedLowSafety : REAL;
   AdvancedHighSafety : REAL;
   JogSpeedPercent : DINT;
   AdvancedDefaultTarget : REAL;
END_STRUCT
END_TYPE

TYPE up_ServoAdvanceReturnCommands :
STRUCT
   JogMode : BOOL;
   JogForward : BOOL;
   JogReverse : BOOL;
   StartHomePulse : BOOL;
   HomeServo : BOOL;
   SetReturnedPosition : BOOL;
   SetAdvancedPosition : BOOL;
END_STRUCT
END_TYPE

TYPE up_ServoAdvanceReturnStatus :
STRUCT
   AtHomePosition : BOOL;
   ValidReturnedPosition : BOOL;
   ValidAdvancedPosition : BOOL;
END_STRUCT
END_TYPE

TYPE up_SpindleServoCommands :
STRUCT
   JogMode : BOOL;
   JogForward : BOOL;
   JogReverse : BOOL;
   StartHomePulse : BOOL;
   HomeSpindleServo : BOOL;
   GoToOrientAngle : BOOL;
   GoToZeroDegrees : BOOL;
   GoToTestAngle : BOOL;
   GoTo180Degrees : BOOL;
   GoToRimChangeAngle : BOOL;
   GoToRimUnlockAngle : BOOL;
END_STRUCT
END_TYPE

TYPE up_SpindleServoStatus :
STRUCT
   AtHomePosition : BOOL;
   ZeroSpeed : BOOL;
   AtOrientAngle : BOOL;
   AtZeroDegrees : BOOL;
   AtTestAngle : BOOL;
   At180Degrees : BOOL;
   AtRimChangeAngle : BOOL;
   AtRimUnlockAngle : BOOL;
   AtUpperToolingAngle : BOOL;
END_STRUCT
END_TYPE

TYPE up_Style :
STRUCT
   Spare1 : BOOL;
   Spare2 : BOOL;
   WriteRequest : SINT;
   WriteSetup : SINT;
   WriteComplete : SINT;
   Clear : SINT;
   Number : BOOL[256];
   NoOperation : BOOL;
   ValidStyle : BOOL;
   InvalidStyle : BOOL;
END_STRUCT
END_TYPE

TYPE up_TransferGripper :
STRUCT
   Command : up_TransferGripperCommands;
   Status : up_TransferGripperStatus;
   EnableMotion : BOOL;
   OpenedTargetIsValid : BOOL;
   ClosedTargetIsValid : BOOL;
   OpenedPositionTarget : DINT;
   OpenedLowLimit : REAL;
   OpenedHighLimit : REAL;
   OpenedLowSafety : DINT;
   OpenedHighSafety : DINT;
   ClosedPositionTarget : DINT;
   ClosedLowLimit : REAL;
   ClosedHighLimit : REAL;
   ClosedLowSafety : DINT;
   ClosedHighSafety : DINT;
   JogSpeedPercent : DINT;
END_STRUCT
END_TYPE

TYPE up_TransferGripperCommands :
STRUCT
   JogMode : BOOL;
   JogGripperClosed : BOOL;
   JogGripperOpen : BOOL;
   StartHomePulse : BOOL;
   HomeServo : BOOL;
   SetGripperOpenedPosition : BOOL;
   SetGripperClosedPosition : BOOL;
END_STRUCT
END_TYPE

TYPE up_TransferGripperStatus :
STRUCT
   AtHomePosition : BOOL;
   ValidOpenPosition : BOOL;
   ValidClosedPosition : BOOL;
END_STRUCT
END_TYPE

TYPE up_UpperRimServo :
STRUCT
   Command : up_UpperRimServoCommands;
   Status : up_UpperRimServoStatus;
   EnableMotion : BOOL;
   RaisedPositionTargetIsValid : BOOL;
   LockPositionTargetIsValid : BOOL;
   ChangerPositionTargetIsValid : BOOL;
   Join1PositionTargetisValid : BOOL;
   Join2PositionTargetIsValid : BOOL;
   RaisedPositionTarget : REAL;
   Step1Target : REAL;
   LockPositionTarget : REAL;
   LockPositionHighLimit : REAL;
   LockPositionLowLimit : REAL;
   ChangerPosiitonTarget : REAL;
   ChangerPositionHighLimit : REAL;
   ChangerPositionLowLimit : REAL;
   Join1PositionTarget : REAL;
   Join1PositionHighLimit : REAL;
   Join1PositionLowLimit : REAL;
   Join2PositionTarget : REAL;
   Join2PositionHighLimit : REAL;
   Join2PositionLowLimit : REAL;
   JogSpeedPercent : DINT;
END_STRUCT
END_TYPE

TYPE up_UpperRimServoCommands :
STRUCT
   JogMode : BOOL;
   JogToolingDowm : BOOL;
   JogToolingUp : BOOL;
   StartHomePulse : BOOL;
   HomeToolingServo : BOOL;
   Set_RaisedPosition : BOOL;
   Set_RimStep1Position : BOOL;
   Set_ChangerPosition : BOOL;
   Set_Join1Position : BOOL;
   Set_Join2Position : BOOL;
END_STRUCT
END_TYPE

TYPE up_UpperRimServoStatus :
STRUCT
   AtHomePosition : BOOL;
   ValidRaisedPosition : BOOL;
   ValidRimStep1Position : BOOL;
   ValidChangerPosition : BOOL;
   ValidJoin1Position : BOOL;
   ValidJoin2Position : BOOL;
END_STRUCT
END_TYPE

TYPE up_Utilities :
STRUCT
   OutputPower : BOOL;
   MainAirPresFltMem : BOOL;
   HydPresFltMem : BOOL;
   ZeroAirPresFltMem : BOOL;
   InflateAirPresFltMem : BOOL;
   MainAirPresOK : TIMER;
   HydPresOK : TIMER;
   InflateAirPresOK : TIMER;
   ZeroAirPresOK : TIMER;
END_STRUCT
END_TYPE

TYPE z_Data :
STRUCT
   Present : BOOL;
   ToPrevDataRcvd : BOOL;
   ToNextDataRcvd : BOOL;
   SeqNumSuffix : SINT;
   BuildStatus : INT;
   Options : INT[8];
   Style : DINT;
   VID : DINT;
   SeqNum : DINT;
   Carrier : DINT;
END_STRUCT
END_TYPE

TYPE z_HMIStylePBs :
STRUCT
   Read : BOOL;
   Write : BOOL;
   Sync : BOOL;
   Clear : BOOL;
   Cancel : BOOL;
   Overview : BOOL;
   Spare : BOOL;
END_STRUCT
END_TYPE

TYPE za_Action :
STRUCT
   Comp : BOOL;
   ProcComp : BOOL;
   Auto : BOOL;
   AutoSetup : BOOL;
   Clear : BOOL;
   ClrSetup : BOOL;
   OutPwr : BOOL;
   Cmd : BOOL;
   Out : BOOL;
   Mem : BOOL;
   PB : BOOL;
   FLT : BOOL;
   Active : BOOL;
   EnableSkip : BOOL;
   EnableBypass : BOOL;
   Bypassed : BOOL;
   Prompt : BOOL;
   OutPwrPrompt : BOOL;
   Setup1 : BOOL;
   Setup2 : BOOL;
   Setup3 : BOOL;
   Setup4 : BOOL;
   AntiRept : BOOL;
   OneShot : BOOL;
   FltCheck : BOOL;
   RecipeEnable : BOOL;
   Text : DINT;
   StatusType : DINT;
   TMR : TIMER;
   Dwell : TIMER;
END_STRUCT
END_TYPE

TYPE zz_StaMode :
STRUCT
   AutoReqAntiRpt : BOOL;
   AutoRdy : BOOL;
   Auto : BOOL;
   ExtrnAutoRdy : BOOL;
   Man : BOOL;
   Tryout : BOOL;
   ByPass : BOOL;
END_STRUCT
END_TYPE

VAR_GLOBAL   (* controller tags *)
   AfterPause : BOOL;
   APOut : BOOL;
   DoNothing : BOOL;
   ECR : BOOL;   // Emergency Control Relay
   EixtPB : BOOL := 1;
   EmergencyPB : BOOL := 1;
   Exit_SEQ : BOOL;
   Exit_SEQONS : BOOL;
   Exit_SEQONS1 : BOOL;
   indicate : DINT := 38;
        .5   // To HMI Indicate Sequence Resume Mode
        .4   // To HMI Indicate Sequence Pause Mode
        .3   // To HMI Indicate Sequence Stop Mode
        .2   // To HMI Indicate Sequence Start Mode
        .1   // To HMI Indicate Master Control Relay On
        .0   // To HMI Indicate EStop Relay On
   LastWord : DINT := 2335;
   MasterStart : BOOL;
   MasterStartCommand : BOOL := 1;
   MasterStop : BOOL;
   MCR : BOOL := 1;   // Master Control Relay
   N10 : DINT[32] := ([0] := 1);
   NotContinue : BOOL;
   OutWord : DINT;
   SCR : BOOL := 1;   // Sequence Control Relay
   SEQCon : BOOL;
   SeQCount : DINT := 1;
   SEQPause : BOOL;
   SeqPausePB : BOOL := 1;
   SEQResume : BOOL := 1;
   SeqRunOk : BOOL;
   SPR : BOOL;   // Sequence Pause Relay
   SRR : BOOL := 1;   // Sequence Resume Relay
   SSR : BOOL;   // Stop Sequence Relay
   StartPBCom : BOOL;
   StartSeq : BOOL;
   StopSeq : BOOL := 1;
END_VAR

PROGRAM MainProgram   (* main routine MainRoutine *)
VAR
   Action_000 : SFC_ACTION := (Status := 16#c020_0000, A := 1, Q := 1, PauseTimer := 1, Count := 147);
   Action_001 : SFC_ACTION := (Status := 16#c020_0000, A := 1, Q := 1, PauseTimer := 1, Count := 147);
   Action_002 : SFC_ACTION := (Status := 16#0020_0000, PauseTimer := 1, Count := 146);
   Action_003 : SFC_ACTION := (Status := 16#0020_0000, PauseTimer := 1, Count := 146);
   Action_004 : SFC_ACTION := (Status := 16#0020_0000, PauseTimer := 1, Count := 146);
   Action_005 : SFC_ACTION := (Status := 16#0020_0000, PauseTimer := 1, Count := 146);
   Action_006 : SFC_ACTION := (Status := 16#0020_0000, PauseTimer := 1, Count := 146);
   Action_007 : SFC_ACTION := (Status := 16#0020_0000, PauseTimer := 1, Count := 146);
   Action_008 : SFC_ACTION := (Status := 16#0020_0000, PauseTimer := 1, Count := 146);
   Action_009 : SFC_ACTION := (Status := 16#0020_0000, PauseTimer := 1, Count := 146);
   Action_010 : SFC_ACTION := (Status := 16#0020_0000, PauseTimer := 1, Count := 146);
   Action_011 : SFC_ACTION := (Status := 16#0020_0000, PauseTimer := 1, Count := 146);
   Action_012 : SFC_ACTION := (Status := 16#0020_0000, PauseTimer := 1, Count := 146);
   Continue : BOOL := 1;
   Count : DINT := 1;
   Step_000 : SFC_STEP := (Status := 16#0820_0201, DN := 1, PauseTimer := 1, PRE := 500, T := 500, TMax := 21046, Count := 147);
   Step_001 : SFC_STEP := (Status := 16#0820_0001, DN := 1, PauseTimer := 1, PRE := 500, T := 500, TMax := 690958, Count := 146);
   Step_002 : SFC_STEP := (Status := 16#0820_0001, DN := 1, PauseTimer := 1, PRE := 500, T := 500, TMax := 8010, Count := 146);
   Step_003 : SFC_STEP := (Status := 16#0820_0001, DN := 1, PauseTimer := 1, PRE := 500, T := 500, TMax := 220188, Count := 146);
   Step_004 : SFC_STEP := (Status := 16#0820_0001, DN := 1, PauseTimer := 1, PRE := 500, T := 500, TMax := 11621, Count := 146);
   Step_005 : SFC_STEP := (Status := 16#0820_0001, DN := 1, PauseTimer := 1, PRE := 500, T := 500, TMax := 1300357, Count := 146);
   Step_006 : SFC_STEP := (Status := 16#0820_0001, DN := 1, PauseTimer := 1, PRE := 500, T := 500, TMax := 23739, Count := 146);
   Step_007 : SFC_STEP := (Status := 16#0820_0001, DN := 1, PauseTimer := 1, PRE := 500, T := 500, TMax := 2969, Count := 146);
   Step_008 : SFC_STEP := (Status := 16#0820_0001, DN := 1, PauseTimer := 1, PRE := 500, T := 500, TMax := 6700, Count := 146);
   Step_009 : SFC_STEP := (Status := 16#0820_0001, DN := 1, PauseTimer := 1, PRE := 500, T := 500, TMax := 501, Count := 146);
   Step_010 : SFC_STEP := (Status := 16#0820_0001, DN := 1, PauseTimer := 1, PRE := 500, T := 500, TMax := 196095, Count := 146);
   Step_011 : SFC_STEP := (Status := 16#0820_0001, DN := 1, PauseTimer := 1, PRE := 500, T := 500, TMax := 3830682, Count := 146);
   Step_012 : SFC_STEP := (Status := 16#0020_0001, PauseTimer := 1, PRE := 500, TMax := 1, Count := 146);
   Tran_000 : BOOL;
   Tran_001 : BOOL := 1;
   Tran_002 : BOOL := 1;
   Tran_003 : BOOL := 1;
   Tran_004 : BOOL := 1;
   Tran_005 : BOOL := 1;
   Tran_006 : BOOL := 1;
   Tran_007 : BOOL := 1;
   Tran_008 : BOOL := 1;
   Tran_009 : BOOL := 1;
   Tran_010 : BOOL := 1;
   Tran_011 : BOOL := 1;
   Tran_012 : BOOL := 1;
   Tran_013 : BOOL;
   Tran_014 : BOOL;
   Tran_015 : BOOL;
   Tran_016 : BOOL;
   Tran_017 : BOOL;
   Tran_018 : BOOL;
   Tran_019 : BOOL;
   Tran_020 : BOOL;
   Tran_021 : BOOL;
   Tran_022 : BOOL;
   Tran_023 : BOOL;
   Tran_024 : BOOL;
   Tran_025 : BOOL;
END_VAR

ROUTINE A000Conditions   (* ladder *)
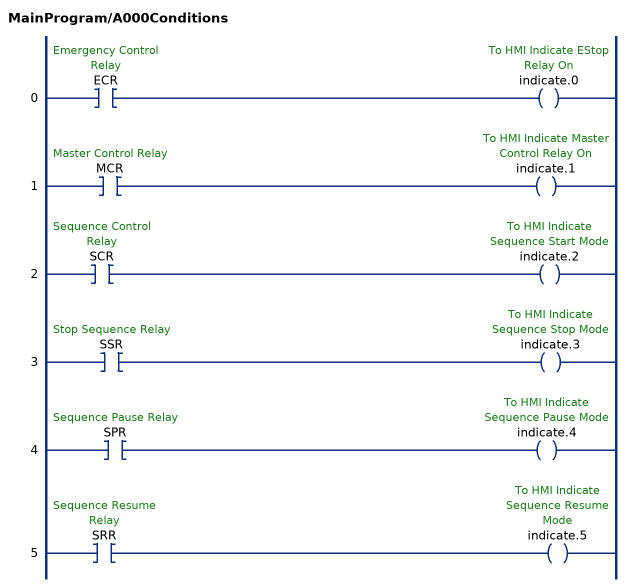
   0: XIC(ECR)OTE(indicate.0);
   1: XIC(MCR)OTE(indicate.1);
   2: XIC(SCR)OTE(indicate.2);
   3: XIC(SSR)OTE(indicate.3);
   4: XIC(SPR)OTE(indicate.4);
   5: XIC(SRR)OTE(indicate.5);
END_ROUTINE

ROUTINE MainRoutine   (* ladder *)
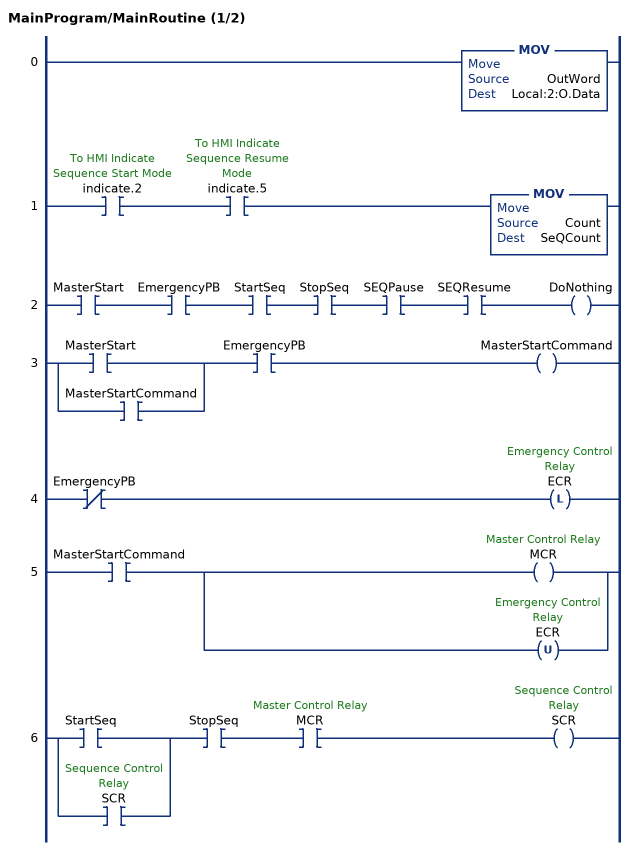
   0: MOV(OutWord,Local:2:O.Data);
   1: XIC(indicate.2)XIC(indicate.5)MOV(Count,SeQCount);
   2: XIC(MasterStart)XIC(EmergencyPB)XIC(StartSeq)XIC(StopSeq)XIC(SEQPause)XIC(SEQResume)OTE(DoNothing);
   3: [XIC(MasterStart) ,XIC(MasterStartCommand) ]XIC(EmergencyPB)OTE(MasterStartCommand);
   4: XIO(EmergencyPB)OTL(ECR);
   5: XIC(MasterStartCommand)[OTE(MCR) ,OTU(ECR) ];
   6: [XIC(StartSeq) ,XIC(SCR) ]XIC(StopSeq)XIC(MCR)OTE(SCR);
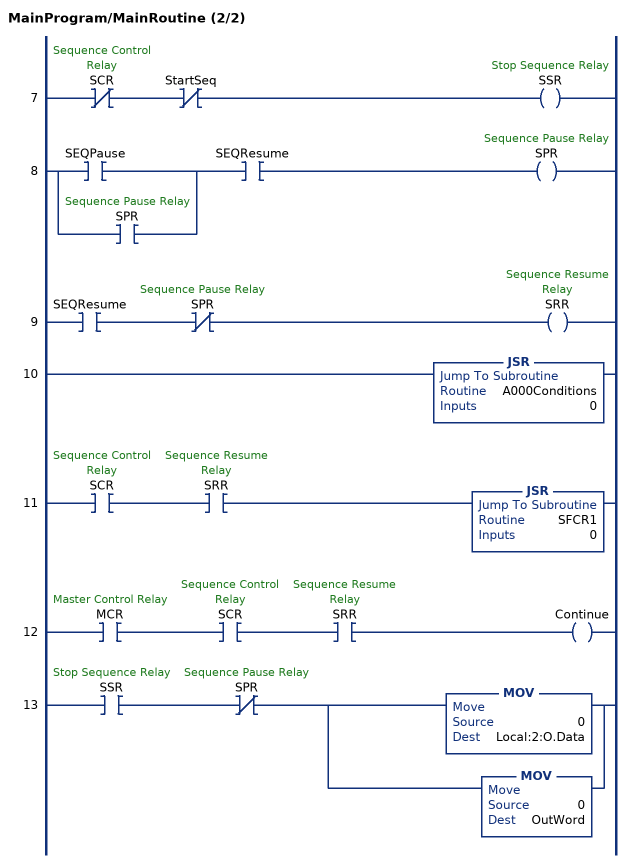
   7: XIO(SCR)XIO(StartSeq)OTE(SSR);
   8: [XIC(SEQPause) ,XIC(SPR) ]XIC(SEQResume)OTE(SPR);
   9: XIC(SEQResume)XIO(SPR)OTE(SRR);
   10: JSR(A000Conditions,0);
   11: XIC(SCR)XIC(SRR)JSR(SFCR1,0);
   12: XIC(MCR)XIC(SCR)XIC(SRR)OTE(Continue);
   13: XIC(SSR)XIO(SPR)[MOV(0,Local:2:O.Data) ,MOV(0,OutWord) ];
END_ROUTINE

ROUTINE SFCR1   (* sequential function chart *)
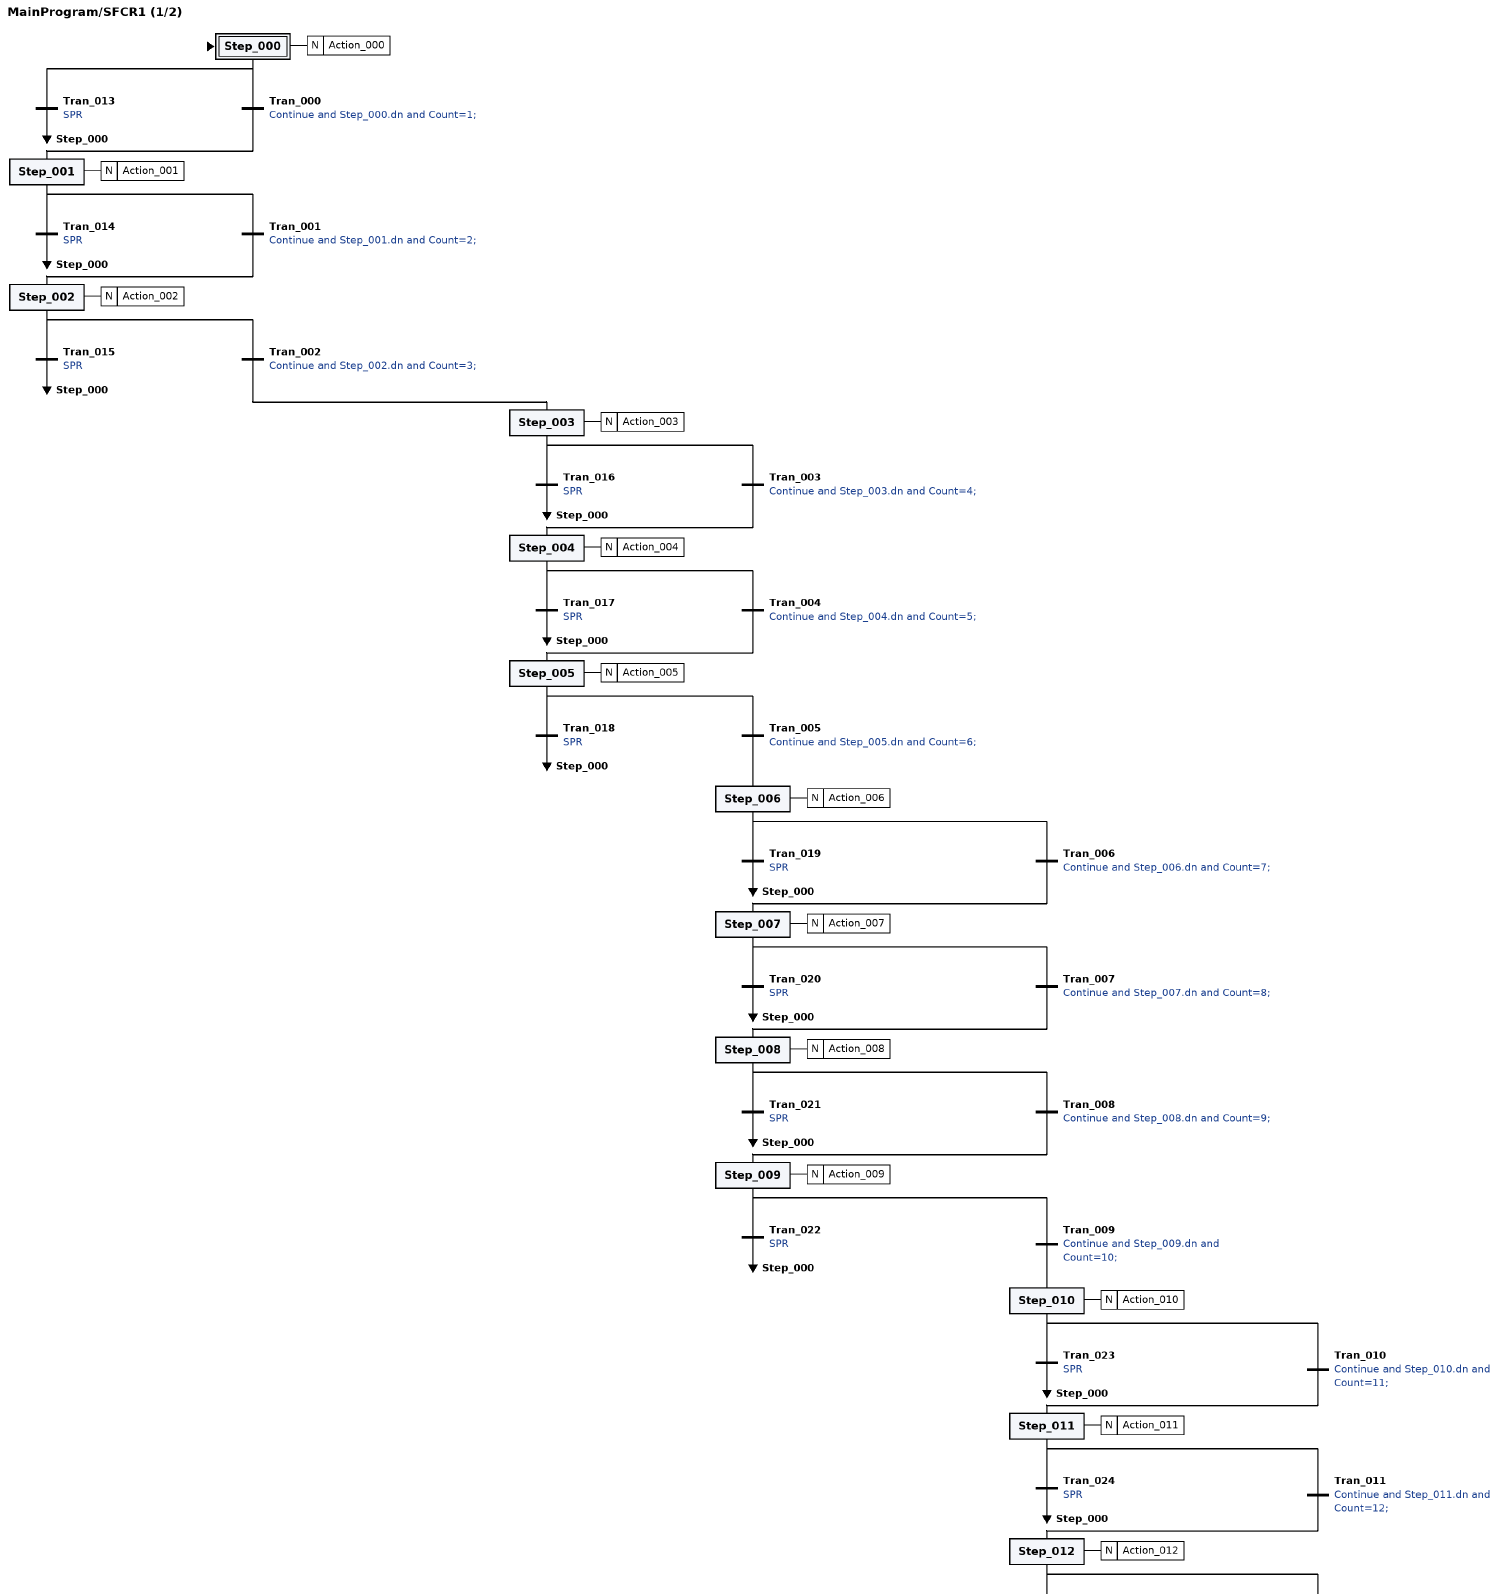
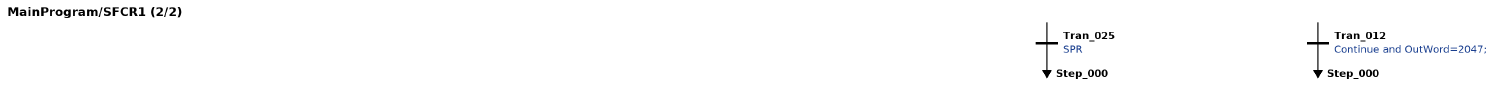
   STEP Step_003:
      ACTION Action_003 (N):
         OutWord :=7;
         Count :=4;
      END_ACTION
   END_STEP
   INITIAL_STEP Step_000:
      ACTION Action_000 (N):
         OutWord :=0;
         Count :=1;
         
         
      END_ACTION
   END_STEP
   STEP Step_006:
      ACTION Action_006 (N):
         OutWord :=63;
         Count :=7;
      END_ACTION
   END_STEP
   TRANSITION Tran_016 FROM Step_003 TO Step_000
      := SPR
         
   END_TRANSITION
   TRANSITION Tran_003 FROM Step_003 TO Step_004
      := Continue and Step_003.dn and Count=4;
   END_TRANSITION
   STEP Step_010:
      ACTION Action_010 (N):
         OutWord :=1023;
         Count :=11;
         
      END_ACTION
   END_STEP
   TRANSITION Tran_013 FROM Step_000 TO Step_000
      := SPR
         
   END_TRANSITION
   TRANSITION Tran_000 FROM Step_000 TO Step_001
      := Continue and Step_000.dn and   Count=1;
   END_TRANSITION
   TRANSITION Tran_019 FROM Step_006 TO Step_000
      := SPR
         
   END_TRANSITION
   TRANSITION Tran_006 FROM Step_006 TO Step_007
      := Continue and Step_006.dn and Count=7;
   END_TRANSITION
   STEP Step_001:
      ACTION Action_001 (N):
         OutWord :=1;
         Count :=2;
      END_ACTION
   END_STEP
   STEP Step_004:
      ACTION Action_004 (N):
         OutWord :=15;
         Count :=5;
      END_ACTION
   END_STEP
   STEP Step_007:
      ACTION Action_007 (N):
         OutWord :=127;
         Count :=8;
      END_ACTION
   END_STEP
   TRANSITION Tran_023 FROM Step_010 TO Step_000
      := SPR
         
   END_TRANSITION
   TRANSITION Tran_010 FROM Step_010 TO Step_011
      := Continue and Step_010.dn and Count=11;
   END_TRANSITION
   TRANSITION Tran_014 FROM Step_001 TO Step_000
      := SPR
         
   END_TRANSITION
   TRANSITION Tran_017 FROM Step_004 TO Step_000
      := SPR
         
   END_TRANSITION
   TRANSITION Tran_004 FROM Step_004 TO Step_005
      := Continue and Step_004.dn and Count=5;
   END_TRANSITION
   STEP Step_011:
      ACTION Action_011 (N):
         OutWord :=2047;
         Count :=12;
      END_ACTION
   END_STEP
   TRANSITION Tran_001 FROM Step_001 TO Step_002
      := Continue and Step_001.dn and Count=2;
   END_TRANSITION
   STEP Step_005:
      ACTION Action_005 (N):
         OutWord :=31;
         Count :=6;
      END_ACTION
   END_STEP
   TRANSITION Tran_020 FROM Step_007 TO Step_000
      := SPR
         
   END_TRANSITION
   TRANSITION Tran_007 FROM Step_007 TO Step_008
      := Continue and Step_007.dn and Count=8;
   END_TRANSITION
   STEP Step_002:
      ACTION Action_002 (N):
         OutWord :=3;
         Count :=3;
      END_ACTION
   END_STEP
   STEP Step_008:
      ACTION Action_008 (N):
         OutWord :=255;
         Count :=9;
      END_ACTION
   END_STEP
   TRANSITION Tran_024 FROM Step_011 TO Step_000
      := SPR
         
   END_TRANSITION
   TRANSITION Tran_011 FROM Step_011 TO Step_012
      := Continue and Step_011.dn and Count=12;
   END_TRANSITION
   TRANSITION Tran_018 FROM Step_005 TO Step_000
      := SPR
         
   END_TRANSITION
   TRANSITION Tran_005 FROM Step_005 TO Step_006
      := Continue and Step_005.dn and Count=6;
   END_TRANSITION
   STEP Step_012:
      ACTION Action_012 (N):
         OutWord :=2047;
      END_ACTION
   END_STEP
   TRANSITION Tran_015 FROM Step_002 TO Step_000
      := SPR
         
   END_TRANSITION
   TRANSITION Tran_002 FROM Step_002 TO Step_003
      := Continue and Step_002.dn and Count=3;
   END_TRANSITION
   TRANSITION Tran_021 FROM Step_008 TO Step_000
      := SPR
         
   END_TRANSITION
   TRANSITION Tran_008 FROM Step_008 TO Step_009
      := Continue and Step_008.dn and Count=9;
   END_TRANSITION
   STEP Step_009:
      ACTION Action_009 (N):
         OutWord :=511;
         Count :=10;
      END_ACTION
   END_STEP
   TRANSITION Tran_025 FROM Step_012 TO Step_000
      := SPR
         
   END_TRANSITION
   TRANSITION Tran_012 FROM Step_012 TO Step_000
      := Continue and OutWord=2047;
   END_TRANSITION
   TRANSITION Tran_022 FROM Step_009 TO Step_000
      := SPR
         
   END_TRANSITION
   TRANSITION Tran_009 FROM Step_009 TO Step_010
      := Continue and Step_009.dn and Count=10;
   END_TRANSITION
END_ROUTINE

ROUTINE SFCR2   (* sequential function chart *)
END_ROUTINE
END_PROGRAM
